// TwinCAT 3 PLC project PLCProgram
// ProgramVersion: 3.1.4024.0
// libraries:
//   Tc2_Standard, * (Beckhoff Automation GmbH)
//   Tc2_System, * (Beckhoff Automation GmbH)
//   Tc2_Utilities, * (Beckhoff Automation GmbH)
//   Tc3_Database, * (Beckhoff Automation GmbH)
//   Tc3_Module, * (Beckhoff Automation GmbH)
// project tree:
//   / PlcTask.TcTTO
//   POUs/ AutoLogData.TcPOU, MAIN.TcPOU
// real-time tasks:
//   TASK PlcTask: cycle T#10ms, priority 20, ADS port 350

CONFIGURATION PLCProgram
    RESOURCE PLC ON TwinCAT3
        TASK PlcTask(INTERVAL := T#10ms, PRIORITY := 20);
        PROGRAM MAIN WITH PlcTask : MAIN;
    END_RESOURCE
END_CONFIGURATION

// ---- POUs/MAIN.TcPOU
PROGRAM MAIN
VAR
	
END_VAR

//Auto Logging
AutoLogData();

END_PROGRAM

// ---- POUs/AutoLogData.TcPOU
PROGRAM AutoLogData
VAR	

	(* Auto Log FB *)	
	fbPLCDBAutoLog    : FB_PLCDBAutoLogEvt(sNetID:='', tTimeout := T#5S);
	
	// Auto Log Group Status
    bError            : BOOL; 
    aAutologGrpStatus : ARRAY[0..MAX_CONFIGURATIONS] OF ST_AutoLogGrpStatus;
	
	//Start & Stop Auto Log
	bStopAutoLog: BOOL;
	bStartAutoLog: BOOL;
	bStartedAutoLog: BOOL;
	
	//Start After 1 Mins
	OneMinTimer: TON; 
	InitTimer : BOOL := TRUE;
	
	(* Auto Log System Latency *)
	pulseTimer: TON;         
    pulseOutput: BOOL := FALSE; 
	fbSystemLatency: TC_SysLatency;
	
	iActualLatency: UDINT;
	iMaxLatency: UDINT;

END_VAR

//Auto Log Group Status
IF fbPLCDBAutoLog.Status(tCheckCycle := T#10S, ADR(bError), ADR(aAutologGrpStatus), SIZEOF(aAutologGrpStatus)) THEN
    ; 
END_IF

//Start Auto Log After 1 Mins
OneMinTimer(IN := InitTimer, PT := T#1M);
//Start Auto Log
IF bStartAutoLog OR OneMinTimer.Q THEN
	IF fbPLCDBAutoLog.Start() THEN
		bStartedAutoLog := TRUE;
		bStartAutoLog := FALSE;
		InitTimer := FALSE;
	END_IF;
END_IF

//Stop Auto Log
IF bStopAutoLog THEN
	IF fbPLCDBAutoLog.Stop() THEN
		bStartedAutoLog := FALSE;
		bStopAutoLog:=FALSE;
	END_IF;
END_IF

(* Pulse Generation *)
pulseTimer(IN := TRUE, PT := T#500MS);
IF pulseTimer.Q THEN
    pulseOutput := TRUE;  // Set pulse output to TRUE when timer reaches 500ms
    pulseTimer(IN := FALSE); // Stop the timer
ELSE
    pulseOutput := FALSE; // Set pulse output to FALSE
END_IF

(* Reading System Latency *)
fbSystemLatency(
	NETID:='192.168.1.19.1.1', 
	START:=pulseOutput, 
	TMOUT:=T#1S, 
	BUSY=> , 
	ERR=> , 
	ERRID=> , 
	ACTUAL=>, 
	MAXIMUM=>);
	
IF NOT fbSystemLatency.BUSY THEN
	iActualLatency := fbSystemLatency.ACTUAL;
	iMaxLatency := fbSystemLatency.MAXIMUM;
END_IF

END_PROGRAM
